TYPE stStickerMachine EXTENDS stPimMachineData :
STRUCT
	
END_STRUCT
END_TYPE

(* stored: Version 1.1.0.1, ProductVersion 3.1.4024.13
   DUT stStickerMachine: Id {8a104e91-5cbe-40b6-9b11-087890099057} *)
